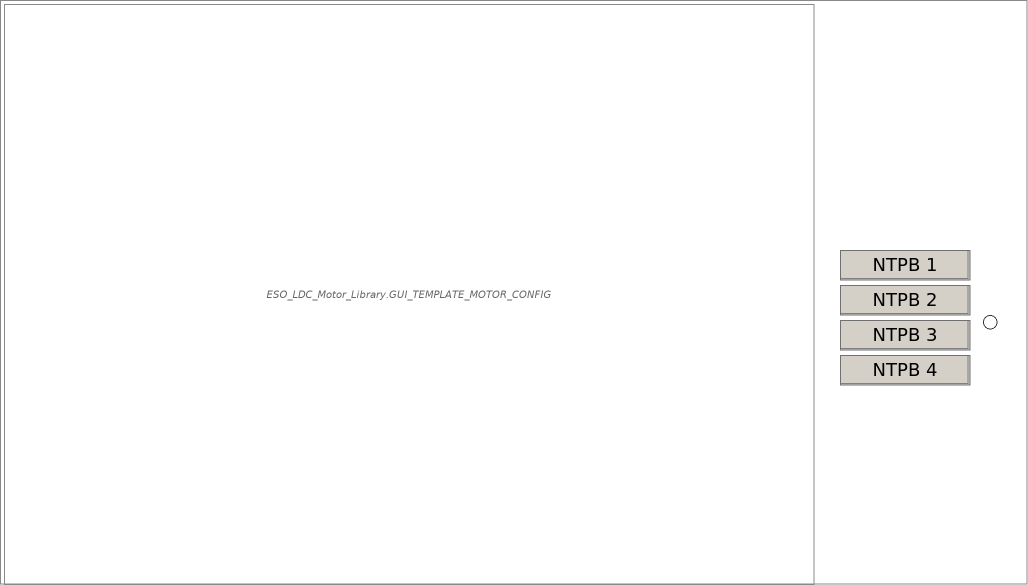
VISUALIZATION GUI_NOTT_TIP_B_CONFIG  // 1028x585
    Frame (4,4 810x581)
        shows ESO_LDC_Motor_Library.GUI_TEMPLATE_MOTOR_CONFIG(m_Instance := MAIN.nott_ics.TipTilt.ptrTipActuatorsB[MAIN.nott_ics.TipTilt.guiTipActuatorsBIndex]^)
    RadioButton (981,252 47x140), variable: MAIN.nott_ics.TipTilt.guiTipActuatorsBIndex-1
        Areas[0]: Text=Radiobutton
        Areas[1]: Text=Radiobutton
    Button (840,250 130x30), "NTPB 1"
        OnMouseClick: execute { MAIN.nott_ics.TipTilt.guiTipActuatorsBIndex := 1; }
    Button (840,285 130x30), "NTPB 2"
        OnMouseClick: execute { MAIN.nott_ics.TipTilt.guiTipActuatorsBIndex := 2; }
    Button (840,320 130x30), "NTPB 3"
        OnMouseClick: execute { MAIN.nott_ics.TipTilt.guiTipActuatorsBIndex := 3; }
    Button (840,355 130x30), "NTPB 4"
        OnMouseClick: execute { MAIN.nott_ics.TipTilt.guiTipActuatorsBIndex := 4; }
END_VISUALIZATION

(* stored: Version 1.1.0.1, ProductVersion 3.1.4024.12
   Visu GUI_NOTT_TIP_B_CONFIG: Id {c9f02df2-0666-4ffb-85d0-aaebe5316884} *)
